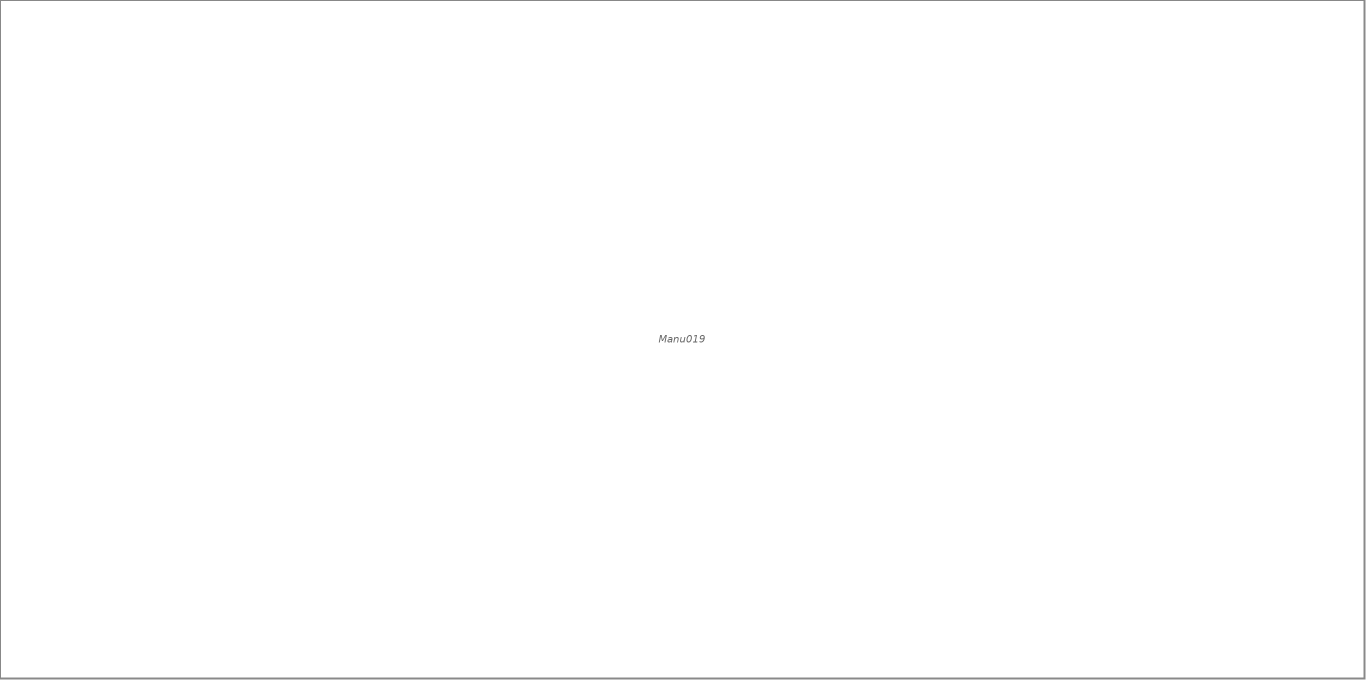
VISUALIZATION Aba_Manu  // 1366x680
    TabControl (0,0 1364x678)
        shows Manu019()
        shows Manu020()
        shows Manu021()
        [0]: TabTitle=203/019
        [1]: TabTitle=203/020
        [2]: TabTitle=203/021
END_VISUALIZATION

(* stored: Version 1.1.0.1, ProductVersion 3.1.4024.12
   Visu Aba_Manu: Id {f4ae9aaa-869f-4226-819b-7cf6702bd561} *)
